FUNCTION LINEAR_LUT : REAL
VAR_INPUT
	rInput:REAL;
END_VAR

VAR_IN_OUT	
	XCol,YCol: ARRAY[*] OF REAL;
END_VAR

VAR
	i,Array1st,ArrayLast: DINT;
	XIncrement:REAL;
END_VAR

Array1st:= LOWER_BOUND(XCol,1);
ArrayLast:= UPPER_BOUND(XCol,1);

IF rInput<= Xcol[Array1st] THEN
	LINEAR_LUT:=YCol[Array1st];
ELSIF rInput>= XCol[ArrayLast] THEN
	LINEAR_LUT:=YCol[ArrayLast];
ELSE
	FOR i:=Array1st TO ArrayLast-1 DO
		IF rInput >= XCol[i] THEN
			XIncrement:= XCol[i+1]-XCol[i];
			IF XIncrement=0 THEN
				LINEAR_LUT:=YCol[i];
			ELSE	
				LINEAR_LUT:=YCol[i]+(rInput-Xcol[i])*(YCol[i+1]-YCol[i])/XIncrement;
				RETURN;
			END_IF;
		END_IF
	END_FOR
END_IF

END_FUNCTION

(* stored: Version 1.1.0.1, ProductVersion 3.1.4024.6
   POU LINEAR_LUT: Id {68eefe84-1122-4026-abe3-d86d7284dda4}, SpecialFunc None *)
